// Mitsubishi GX Works2 project: Conveyor1   PLC: Q02U

PROGRAM MAIN
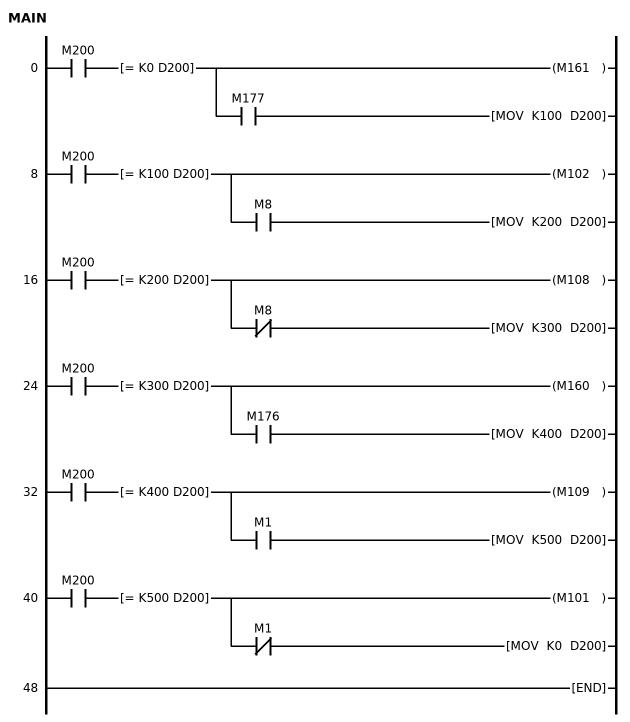
0     LD      M200
      AND=    K0 D200
      OUT     M161
      AND     M177
      MOV     K100 D200
8     LD      M200
      AND=    K100 D200
      OUT     M102
      AND     M8
      MOV     K200 D200
16    LD      M200
      AND=    K200 D200
      OUT     M108
      ANI     M8
      MOV     K300 D200
24    LD      M200
      AND=    K300 D200
      OUT     M160
      AND     M176
      MOV     K400 D200
32    LD      M200
      AND=    K400 D200
      OUT     M109
      AND     M1
      MOV     K500 D200
40    LD      M200
      AND=    K500 D200
      OUT     M101
      ANI     M1
      MOV     K0 D200
48    END
END_PROGRAM

PROGRAM INPUT
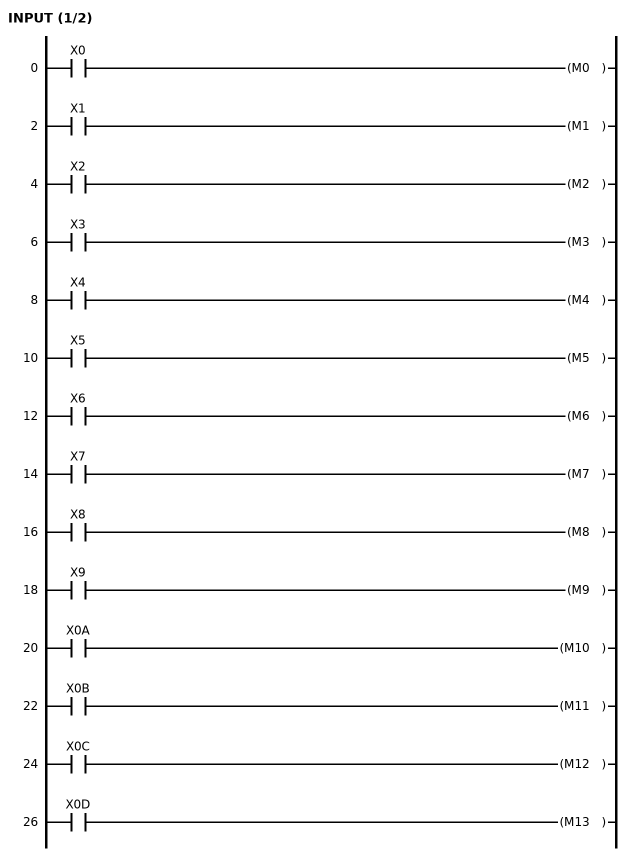
0     LD      X0
      OUT     M0
2     LD      X1
      OUT     M1
4     LD      X2
      OUT     M2
6     LD      X3
      OUT     M3
8     LD      X4
      OUT     M4
10    LD      X5
      OUT     M5
12    LD      X6
      OUT     M6
14    LD      X7
      OUT     M7
16    LD      X8
      OUT     M8
18    LD      X9
      OUT     M9
20    LD      X0A
      OUT     M10
22    LD      X0B
      OUT     M11
24    LD      X0C
      OUT     M12
26    LD      X0D
      OUT     M13
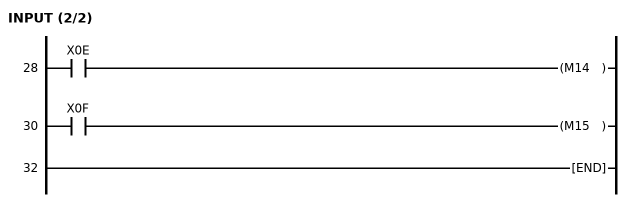
28    LD      X0E
      OUT     M14
30    LD      X0F
      OUT     M15
32    END
END_PROGRAM

PROGRAM OUTPUT
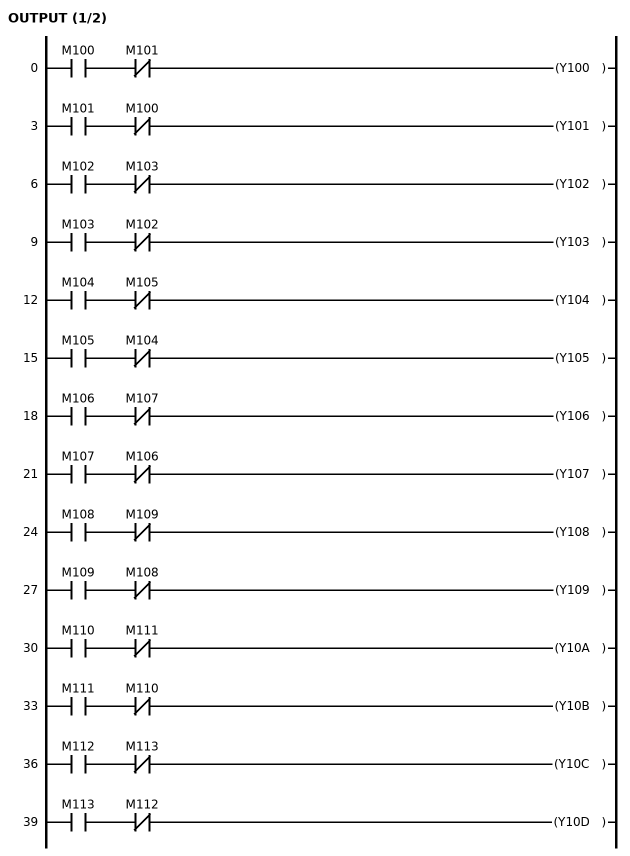
0     LD      M100
      ANI     M101
      OUT     Y100
3     LD      M101
      ANI     M100
      OUT     Y101
6     LD      M102
      ANI     M103
      OUT     Y102
9     LD      M103
      ANI     M102
      OUT     Y103
12    LD      M104
      ANI     M105
      OUT     Y104
15    LD      M105
      ANI     M104
      OUT     Y105
18    LD      M106
      ANI     M107
      OUT     Y106
21    LD      M107
      ANI     M106
      OUT     Y107
24    LD      M108
      ANI     M109
      OUT     Y108
27    LD      M109
      ANI     M108
      OUT     Y109
30    LD      M110
      ANI     M111
      OUT     Y10A
33    LD      M111
      ANI     M110
      OUT     Y10B
36    LD      M112
      ANI     M113
      OUT     Y10C
39    LD      M113
      ANI     M112
      OUT     Y10D
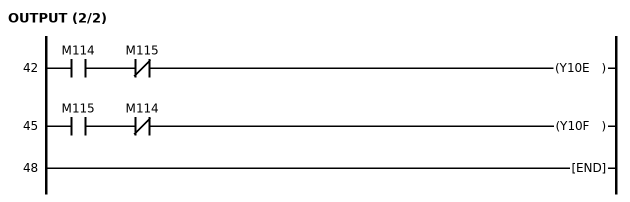
42    LD      M114
      ANI     M115
      OUT     Y10E
45    LD      M115
      ANI     M114
      OUT     Y10F
48    END
END_PROGRAM
